TYPE MotorCommands_typ :
STRUCT
	PowerOn : BOOL;
	Init	: BOOL;
	Home	: BOOL;
	JogPos	: BOOL;
	JogNeg	: BOOL;
	Run		: BOOL;
	Stop	: BOOL;
	ErrorAck: BOOL;
	
END_STRUCT
END_TYPE

(* stored: Version 1.1.0.1, ProductVersion 3.1.4024.15
   DUT MotorCommands_typ: Id {8fd1a564-1925-48ff-a4c5-fe58b1cea691} *)
